Yaskawa INFORM job: POSICAO_MANUTENCAO.JBI

/JOB
//NAME POSICAO_MANUTENCAO
///FOLDERNAME SERVICO
//POS
///NPOS 9,0,9,1,0,1
///TOOL 0
///POSTYPE PULSE
///PULSE
C00000=84296,-111150,-83660,179563,90077,165874
C00001=33886,-105420,-83351,240027,91822,204828
C00002=49988,-101508,-83140,281300,91564,209059
C00003=49988,-101508,-133373,244695,89965,216320
C00004=46570,4014,-163324,185906,70821,212371
C00005=49988,-101508,-133373,244695,89965,216320
C00006=49988,-101508,-83140,281300,91564,209059
C00007=33886,-105420,-83351,240027,91822,204828
C00008=84296,-111150,-83660,179563,90077,165874
EC00000=57494
EC00001=57494
EC00002=57494
EC00003=57494
EC00004=57494
EC00005=57494
EC00006=57494
EC00007=57494
EC00008=57494
P00010=140050,-126820,-84504,14231,87660,95695
EX00010=56001
//INST
///DATE 2022/06/10 15:52
///ATTR SC,RW
///GROUP1 RB1,ST1
NOP
MOVJ P010 EX010 VJ=10.00
MOVJ C00000 EC00000 VJ=10.00
MOVJ C00001 EC00001 VJ=10.00
MOVJ C00002 EC00002 VJ=10.00
MOVJ C00003 EC00003 VJ=10.00
'********************************
MOVJ C00004 EC00004 VJ=10.00 PL=0  //POSICAO DE MANUTENCAO
'********************************
MOVJ C00005 EC00005 VJ=10.00
MOVJ C00006 EC00006 VJ=10.00
MOVJ C00007 EC00007 VJ=10.00
MOVJ C00008 EC00008 VJ=10.00
MOVJ P010 EX010 VJ=10.00
END
